Omron CX-Programmer project NuevoProyecto (CX-Programmer 9.40)

# PLC NuevoPLC1: CQM1 CPU41

## Global symbols (name address type ; comment)
A_mas 100.00 BOOL
B_mas 100.04 BOOL
B_menos 100.05 BOOL
C_mas 100.08 BOOL
C_menos 100.09 BOOL
D_mas 100.12 BOOL
Y_0 100.15 BOOL
a_0 0.00 BOOL
a_1 0.01 BOOL
b_0 0.04 BOOL
b_1 0.05 BOOL
c_0 0.08 BOOL
c_1 0.09 BOOL
flanco_as_a0 16.00 BOOL
flanco_as_c_0 16.01 BOOL
flanco_asc_b0 16.02 BOOL
pe 0.13 BOOL
pm 0.14 BOOL
pp 0.15 BOOL

## Program NuevoPrograma1 (no task)

### Section Sección1

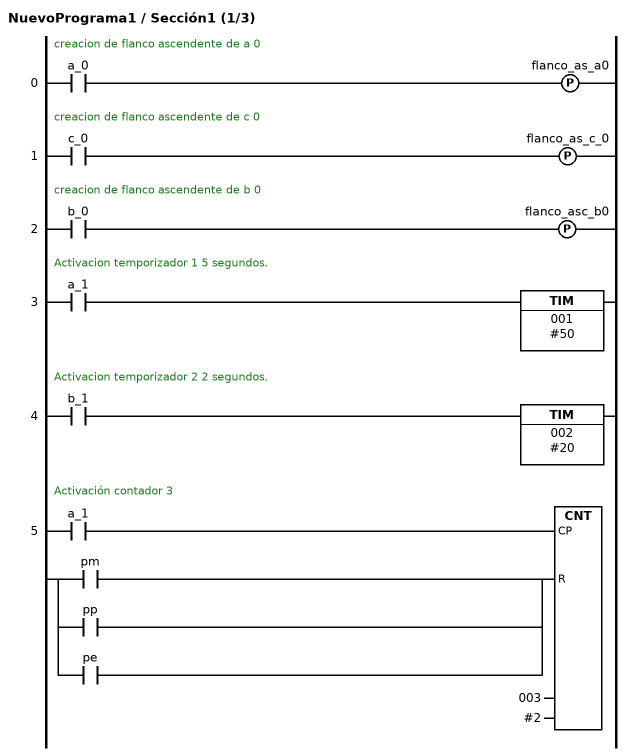
; rung 0: creacion de flanco ascendente de a 0
LD a_0
DIFU(13) flanco_as_a0
; rung 1: creacion de flanco ascendente de c 0
LD c_0
DIFU(13) flanco_as_c_0
; rung 2: creacion de flanco ascendente de b 0
LD b_0
DIFU(13) flanco_asc_b0
; rung 3: Activacion temporizador 1 5 segundos.
LD a_1
TIM 001 #50
; rung 4: Activacion temporizador 2 2 segundos.
LD b_1
TIM 002 #20
; rung 5: Activación contador 3
LD a_1
LD pm
OR pp
OR pe
CNT 003 #2

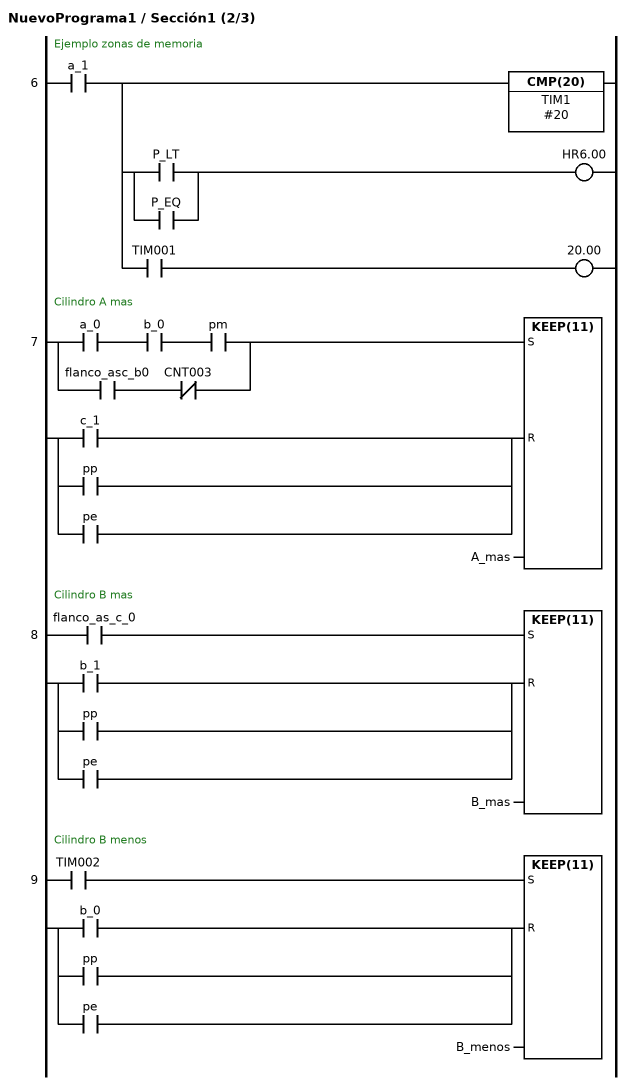
; rung 6: Ejemplo zonas de memoria
LD a_1
OUT TR0
CMP(20) TIM1 #20
LD P_LT
OR P_EQ
ANDLD
OUT HR6.00
LD TR0
AND TIM001
OUT 20.00
; rung 7: Cilindro A mas
LD a_0
AND b_0
AND pm
LD flanco_asc_b0
ANDNOT CNT003
ORLD
LD c_1
OR pp
OR pe
KEEP(11) A_mas
; rung 8: Cilindro B mas
LD flanco_as_c_0
LD b_1
OR pp
OR pe
KEEP(11) B_mas
; rung 9: Cilindro B menos
LD TIM002
LD b_0
OR pp
OR pe
KEEP(11) B_menos

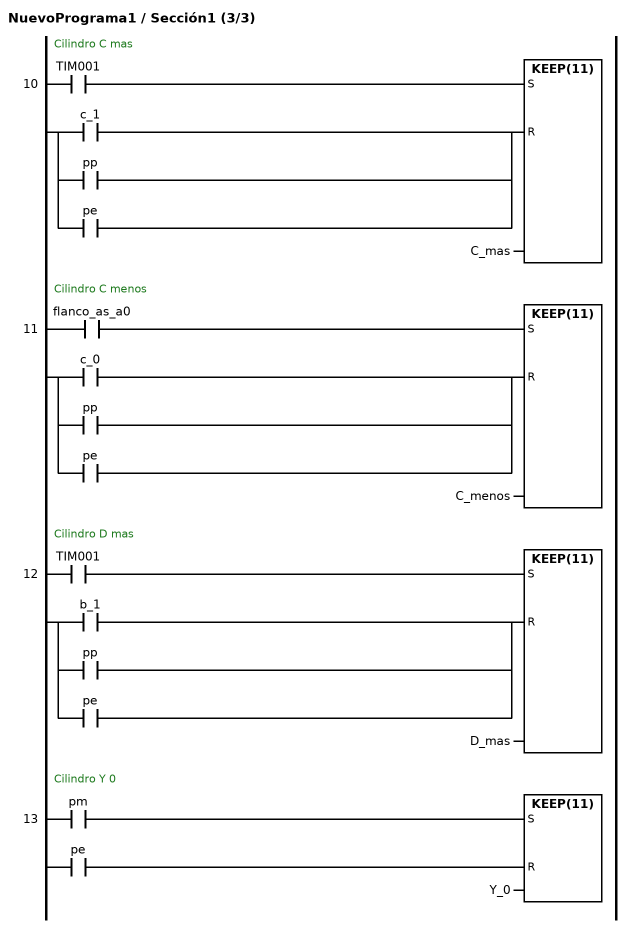
; rung 10: Cilindro C mas
LD TIM001
LD c_1
OR pp
OR pe
KEEP(11) C_mas
; rung 11: Cilindro C menos
LD flanco_as_a0
LD c_0
OR pp
OR pe
KEEP(11) C_menos
; rung 12: Cilindro D mas
LD TIM001
LD b_1
OR pp
OR pe
KEEP(11) D_mas
; rung 13: Cilindro Y 0
LD pm
LD pe
KEEP(11) Y_0

### Section END
; rung 0
END(01)